// TIA Portal V17 export
// export: Created 2025-08-05T09:35:59.9008922Z, ExportSetting WithDefaults, DisplayName Totally Integrated Automation Portal, DisplayVersion V17, DisplayName TIA Portal Openness, DisplayVersion V17, DisplayName TIA Portal Version Control Interface, DisplayVersion V17, DisplayName SINAMICS Startdrive Advanced, DisplayVersion V17, DisplayName SINAMICS Startdrive G130, G150, S120, S150, SINAMICS MV, S210, DisplayVersion V17, DisplayName SINAMICS Startdrive G110M, G120, G120C, G120D, G120P, G115D, DisplayVersion V17, DisplayName STEP 7 Professional, DisplayVersion V17, DisplayName STEP 7 Safety, DisplayVersion V17, DisplayName WinCC Advanced, DisplayVersion V17
TYPE "typeProDiagEvaluation"
TITLE = ProDiag evaluation / ProDiag Auswertung
// ProDiag evaluation [V 01.00 | Kernel_V2] / ProDiag Auswertung [V 01.00 | Kernel_V2]
// stored: IsFailsafeCompliant false
   STRUCT
      faultInstantStop : Bool;   // Störung sofort Halt steht an / Fault immediate stop pending
      faultNoStop : Bool;   // Störung ohne Stop steht an / Fault without stop pending
      faultInCycleEnd : Bool;   // Störung Halt nach Taktende steht an / Fault stop at end of cycle pending
      faultMachineOut : Bool;   // Störung sofort Halt und Maschine Aus steht an / Fault immediate stop and machine off pending
      faultSequence : Bool;   // Ablaufstörung steht an / Sequence fault pending
      message : Bool;   // Meldung steht an / Message pending
      messageOperatorCall : Bool;   // Meldung mit Bedienerruf steht an / Message with operator call pending
      information : Bool;   // Information steht an / Information pending
      popUp : Bool;   // PopUp steht an / Popup pending
      criteriaAnalysis : Bool;   // Kriterienanalyse steht an / Criteria analysis pending
      plcCodeDisplay : Bool;   // Plc Code Anzeige steht an / PLC code display pending
   END_STRUCT;
END_TYPE
